// TIA Portal V19 export
DATA_BLOCK "AlarmGroup"   // DB1
// stored: InstanceOfName AFB_AlarmF, InstanceOfType FB
"AFB_AlarmF"
   // VAR_OUTPUT
   //    faults : Struct
   //       pending : UDInt := 1;
   //       unackn : UDInt := 71;
   //    END_STRUCT;
   //    warnings : Struct
   //       pending { ExternalAccessible := 'False'; ExternalVisible := 'False'; ExternalWritable := 'False'} : UDInt := 0;
   //       unackn { ExternalAccessible := 'False'; ExternalVisible := 'False'; ExternalWritable := 'False'} : UDInt := 5;
   //    END_STRUCT;
   //    fault : Bool := TRUE;
   //    warning : Bool := FALSE;
   //    siren : Bool := TRUE;
   //    icon : Byte := 16#04;
   // END_VAR
   // VAR
   //    M_TYPE_FAULT : Array[0..8] of Int;
   //    M_TYPE_WARNING : Array[0..2] of Int;
   //    nFault : Struct
   //       Alarm : Array[0..8] of UDInt;
   //       Ackn : Array[0..8] of UDInt;
   //       Siren : Array[0..8] of UDInt;
   //    END_STRUCT;
   //    nWarning : Struct
   //       Alarm : Array[0..2] of UDInt;
   //       Ackn : Array[0..2] of UDInt;
   //       Siren : Array[0..2] of UDInt;
   //    END_STRUCT;
   // END_VAR
BEGIN
   M_TYPE_FAULT[0] := 0;
   M_TYPE_FAULT[1] := 3;
   M_TYPE_FAULT[2] := 0;
   M_TYPE_FAULT[3] := 5;
   M_TYPE_FAULT[4] := 3;
   M_TYPE_FAULT[5] := 0;
   M_TYPE_FAULT[6] := 2;
   M_TYPE_FAULT[7] := 0;
   M_TYPE_FAULT[8] := 1;
   M_TYPE_WARNING[0] := 3;
   M_TYPE_WARNING[1] := 0;
   M_TYPE_WARNING[2] := 1;
   nFault.Alarm[0..5] := 0;
   nFault.Alarm[6] := 1;
   nFault.Alarm[7..8] := 0;
   nFault.Ackn[0] := 0;
   nFault.Ackn[1] := 8;
   nFault.Ackn[2] := 0;
   nFault.Ackn[3] := 13;
   nFault.Ackn[4] := 21;
   nFault.Ackn[5] := 0;
   nFault.Ackn[6] := 16;
   nFault.Ackn[7] := 4;
   nFault.Ackn[8] := 8;
   nFault.Siren[0..5] := 0;
   nFault.Siren[6] := 1;
   nFault.Siren[7..8] := 0;
   nWarning.Alarm[0..2] := 0;
   nWarning.Ackn[0] := 4;
   nWarning.Ackn[1] := 0;
   nWarning.Ackn[2] := 1;
   nWarning.Siren[0..2] := 0;
END_DATA_BLOCK
